(* IEC 61131-3 sources: repolevel_ST_code_completion/dataset/generation_context_ground_truth/three-axis_CNC_motion, 4 files *)

(* ---- FB_TripleAxisHoming.st ---- *)
VAR
	fbHomingX			:	SMC_HOMING;			//X轴回零功能块
	fbHomingY			:	SMC_HOMING;			//Y轴回零功能块
	fbHomingZ			:	SMC_HOMING;			//Z轴回零功能块
	fbDoneXTrig			:	R_TRIG;				//X轴完成上升沿
	fbDoneYTrig			:	R_TRIG;				//Y轴完成上升沿
	fbDoneZTrig			:	R_TRIG;				//Z轴完成上升沿
END_VAR

// X轴回零
fbHomingX(
	bExecute := bExecute,
	bReferenceSwitch := bAxisXRefSwitch,
	fVelocitySlow := fVelocitySlow,
	fVelocityFast := fVelocityFast,
	fAcceleration := fAcceleration,
	fDeceleration := fDeceleration,
	Axis := AxisX
);

// Y轴回零
fbHomingY(
	bExecute := bExecute,
	bReferenceSwitch := bAxisYRefSwitch,
	fVelocitySlow := fVelocitySlow,
	fVelocityFast := fVelocityFast,
	fAcceleration := fAcceleration,
	fDeceleration := fDeceleration,
	Axis := AxisY
);

// Z轴回零
fbHomingZ(
	bExecute := bExecute,
	bReferenceSwitch := bAxisZRefSwitch,
	fVelocitySlow := fVelocitySlow,
	fVelocityFast := fVelocityFast,
	fAcceleration := fAcceleration,
	fDeceleration := fDeceleration,
	Axis := AxisZ
);

// 检测X轴完成
fbDoneXTrig(CLK := fbHomingX.bDone);
IF fbDoneXTrig.Q THEN
	bAxisXHomeOK := TRUE;
END_IF

// 检测Y轴完成
fbDoneYTrig(CLK := fbHomingY.bDone);
IF fbDoneYTrig.Q THEN
	bAxisYHomeOK := TRUE;
END_IF

// 检测Z轴完成
fbDoneZTrig(CLK := fbHomingZ.bDone);
IF fbDoneZTrig.Q THEN
	bAxisZHomeOK := TRUE;
END_IF

// 更新输出状态
bHomeOK := bAxisXHomeOK AND bAxisYHomeOK AND bAxisZHomeOK;
bBusy := fbHomingX.bBusy OR fbHomingY.bBusy OR fbHomingZ.bBusy;

// 错误检查（优先级：X > Y > Z）
IF fbHomingX.bError THEN
	bError := TRUE;
	SMC_ERRORSTRING(ErrorID := fbHomingX.nErrorID, Language := english, SMC_ErrorString => sErrorString);
ELSIF fbHomingY.bError THEN
	bError := TRUE;
	SMC_ERRORSTRING(ErrorID := fbHomingY.nErrorID, Language := english, SMC_ErrorString => sErrorString);
ELSIF fbHomingZ.bError THEN
	bError := TRUE;
	SMC_ERRORSTRING(ErrorID := fbHomingZ.nErrorID, Language := english, SMC_ErrorString => sErrorString);
ELSE
	bError := FALSE;
	sErrorString := 'CNC_NO_ERROR';
END_IF

// 复位逻辑
IF NOT bExecute THEN
	bAxisXHomeOK := FALSE;
	bAxisYHomeOK := FALSE;
	bAxisZHomeOK := FALSE;
	bHomeOK := FALSE;
END_IF

(* ---- FB_TripleAxisPower.st ---- *)
VAR
	fbPowerX		:	MC_POWER;			//X轴电源控制
	fbPowerY		:	MC_POWER;			//Y轴电源控制
	fbPowerZ		:	MC_POWER;			//Z轴电源控制
END_VAR

// X轴电源控制
fbPowerX(
	Enable := bServoEnable,
	bRegulatorOn := bServoEnable,
	bDriveStart := bServoEnable,
	Axis := AxisX
);

// Y轴电源控制
fbPowerY(
	Enable := bServoEnable,
	bRegulatorOn := bServoEnable,
	bDriveStart := bServoEnable,
	Axis := AxisY
);

// Z轴电源控制
fbPowerZ(
	Enable := bServoEnable,
	bRegulatorOn := bServoEnable,
	bDriveStart := bServoEnable,
	Axis := AxisZ
);

// 更新输出状态
bAxisXReady := fbPowerX.Status;
bAxisYReady := fbPowerY.Status;
bAxisZReady := fbPowerZ.Status;
bReady := fbPowerX.Status AND fbPowerY.Status AND fbPowerZ.Status;

// 错误检查（优先级：X > Y > Z）
IF fbPowerX.Error THEN
	bError := TRUE;
	SMC_ERRORSTRING(ErrorID := fbPowerX.ErrorID, Language := english, SMC_ErrorString => sErrorString);
ELSIF fbPowerY.Error THEN
	bError := TRUE;
	SMC_ERRORSTRING(ErrorID := fbPowerY.ErrorID, Language := english, SMC_ErrorString => sErrorString);
ELSIF fbPowerZ.Error THEN
	bError := TRUE;
	SMC_ERRORSTRING(ErrorID := fbPowerZ.ErrorID, Language := english, SMC_ErrorString => sErrorString);
ELSE
	bError := FALSE;
	sErrorString := 'CNC_NO_ERROR';
END_IF

(* ---- FB_TripleAxisReset.st ---- *)
VAR
	fbResetX		:	MC_RESET;			//X轴复位
	fbResetY		:	MC_RESET;			//Y轴复位
	fbResetZ		:	MC_RESET;			//Z轴复位
END_VAR

// X轴复位
fbResetX(
	Execute := bExecute,
	Axis := AxisX
);

// Y轴复位
fbResetY(
	Execute := bExecute,
	Axis := AxisY
);

// Z轴复位
fbResetZ(
	Execute := bExecute,
	Axis := AxisZ
);

// 更新输出状态
bBusy := fbResetX.Busy OR fbResetY.Busy OR fbResetZ.Busy;
bDone := fbResetX.Done AND fbResetY.Done AND fbResetZ.Done;

// 错误检查（优先级：X > Y > Z）
IF fbResetX.Error THEN
	bError := TRUE;
	SMC_ERRORSTRING(ErrorID := fbResetX.ErrorID, Language := english, SMC_ErrorString => sErrorString);
ELSIF fbResetY.Error THEN
	bError := TRUE;
	SMC_ERRORSTRING(ErrorID := fbResetY.ErrorID, Language := english, SMC_ErrorString => sErrorString);
ELSIF fbResetZ.Error THEN
	bError := TRUE;
	SMC_ERRORSTRING(ErrorID := fbResetZ.ErrorID, Language := english, SMC_ErrorString => sErrorString);
ELSE
	bError := FALSE;
	sErrorString := 'CNC_NO_ERROR';
END_IF

(* ---- FB_TripleAxisStop.st ---- *)
VAR
	fbStopX			:	MC_STOP;			//X轴停止
	fbStopY			:	MC_STOP;			//Y轴停止
	fbStopZ			:	MC_STOP;			//Z轴停止
END_VAR

// X轴停止
fbStopX(
	Execute := bExecute,
	Deceleration := rDeceleration,
	Axis := AxisX
);

// Y轴停止
fbStopY(
	Execute := bExecute,
	Deceleration := rDeceleration,
	Axis := AxisY
);

// Z轴停止
fbStopZ(
	Execute := bExecute,
	Deceleration := rDeceleration,
	Axis := AxisZ
);

// 更新输出状态
bBusy := fbStopX.Busy OR fbStopY.Busy OR fbStopZ.Busy;
bDone := fbStopX.Done AND fbStopY.Done AND fbStopZ.Done;

// 错误检查（优先级：X > Y > Z）
IF fbStopX.Error THEN
	bError := TRUE;
	SMC_ERRORSTRING(ErrorID := fbStopX.ErrorID, Language := english, SMC_ErrorString => sErrorString);
ELSIF fbStopY.Error THEN
	bError := TRUE;
	SMC_ERRORSTRING(ErrorID := fbStopY.ErrorID, Language := english, SMC_ErrorString => sErrorString);
ELSIF fbStopZ.Error THEN
	bError := TRUE;
	SMC_ERRORSTRING(ErrorID := fbStopZ.ErrorID, Language := english, SMC_ErrorString => sErrorString);
ELSE
	bError := FALSE;
	sErrorString := 'CNC_NO_ERROR';
END_IF
